{attribute 'linkalways'} 
{attribute 'no_explicit_call' := 'This FB is a CLASS and must be accessed using methods or properties'}
{attribute 'enable_dynamic_creation'}
FUNCTION_BLOCK Node_ContainerType_Vector_DINT EXTENDS Node
VAR
    out : _GUID;
END_VAR

METHOD PUBLIC  Clone : I_Node
VAR
	pNode : POINTER TO Node_ContainerType_Vector_DINT;
END_VAR
pNode := __NEW(Node_ContainerType_Vector_DINT);
Clone := pNode^;
END_METHOD

METHOD FB_init : BOOL
VAR_INPUT
	bInitRetains : BOOL; // if TRUE, the retain variables are initialized (warm start / cold start)
	bInCopyCode : BOOL;  // if TRUE, the instance afterwards gets moved into the copy code (online change)
END_VAR
AddOutput('out', out);
END_METHOD

METHOD PROTECTED OnExecute
out.Value := ContainerType_Vector_DINT;
END_METHOD

END_FUNCTION_BLOCK

(* stored: Version 1.1.0.1, ProductVersion 3.1.4026.17
   POU Node_ContainerType_Vector_DINT: Id {e577397e-b7b4-062f-07e4-ab428c1b2bbe}, SpecialFunc None
   Folder Constructor: Id {8a67873e-ee08-04bd-0147-a6bd9c2f6f47}
   Method Clone: Id {39f70f31-19e2-0186-20b5-954dff2c6a1c}
   Method FB_init: Id {aacd6ed3-6e01-0cb2-1c1f-60b680a6218a}
   Method OnExecute: Id {5f1220a8-0e92-049a-30b1-d0365b5c94b8} *)
